FUNCTION calcTimeDiff : LREAL
VAR_INPUT
	TimeCam : TIMESTRUCT;
	TimeSys : TIMESTRUCT; 
END_VAR
VAR
END_VAR

END_FUNCTION

(* stored: Version 1.1.0.1, ProductVersion 3.1.4024.11
   POU calcTimeDiff: Id {de4b1c24-c107-4cbb-a7f2-3430a4a388b4}, SpecialFunc None *)
